PROGRAM Transporteren_order
VAR
	currentState : Taak_2 := Taak_2.Functie;
	Huidige_tijd: INT ;
	Controleren_tijd: BOOL;
	Wachten: BOOL;
	Inladen_krat: BOOL;
END_VAR

Controleren_tijd :=POU(Huidige_tijd);   

CASE currentState OF
	Taak_2.Functie:
		IF Controleren_tijd = TRUE THEN
			CurrentState := taak_2.inladen;
			Wachten := FALSE;
		ELSIF Controleren_tijd = FALSE THEN
			Wachten := TRUE;
			CurrentState := taak_2.Functie;
		END_IF
	
	Taak_2.Inladen:
		IF Controleren_tijd = TRUE THEN
			Inladen_krat := TRUE;
		ELSIF Controleren_tijd = FALSE THEN
			Wachten:= TRUE;
			CurrentState := taak_2.Functie;
			Inladen_krat := FALSE;
		END_IF
		
			
		
END_CASE

END_PROGRAM

(* stored: Version 1.1.0.1, ProductVersion 3.1.4024.12
   POU Transporteren_order: Id {00baf4e9-3cbf-4d61-b5e6-c471975a92d7}, SpecialFunc None *)
